FUNCTION_BLOCK E_SR (* Event-driven bistable *)
  (* Standard: 61499-1-A.1; Classification: Event Processing *)
  (* Version 0.2, 2003-12-30, JHC, Rockwell Automation, Updated for 61499-1 CDV. *)
  (* Version 0.1, 2001-08-16, JHC, Rockwell Automation, XML version *)
  (* Version 0.0, 1998-04-11, JHC, Rockwell Automation, SRC version *)
  (* Compiler header: package fb.rt.events; *)
  (* Compiler Java IBM VisualAge 3.0 *)
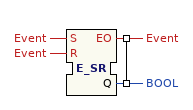
  EVENT_INPUT
    S; (* Set Event *)
    R; (* Reset Event *)
  END_EVENT
  EVENT_OUTPUT
    EO WITH Q; (* Output Event *)
  END_EVENT
  VAR_OUTPUT
    Q : BOOL; (* Current Output State *)
  END_VAR
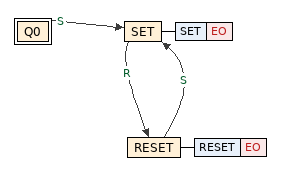
  EC_STATES
    Q0; (* Q is FALSE initially *)
    RESET : RESET -> EO; (* Reset Q and issue EO *)
    SET : SET -> EO; (* Set Q and issue EO *)
  END_STATES
  EC_TRANSITIONS
    Q0 TO SET := S;
    SET TO RESET := R;
    RESET TO SET := S;
  END_TRANSITIONS
  ALGORITHM SET IN ST: (* Set Q *)
Q:=TRUE;
  END_ALGORITHM
  ALGORITHM RESET IN ST: (* Reset Q *)
Q:=FALSE;
  END_ALGORITHM
END_FUNCTION_BLOCK
